		80:	// ABORTING
			// code that is executed only in the first cycle of this state
				IF xStateChange = TRUE THEN
					xStateChange := FALSE;
					iResponse := eResponseReadMalfunctionList.aborting;
					xBusy := FALSE;
					xDone := FALSE;
					xError := FALSE;
					xAborted := TRUE;
				END_IF
			//-----------------------------------------------------------------------------------------------------------
			
			// code that is repeated every cycle in this state
				IF iCurrentValveMode = 63 THEN
					iCommandNumber := 5;	// exit transfer mode
				ELSIF iCurrentValveMode <> 61 AND iCurrentValveMode <> 63 THEN
					iCommandNumber := 6;	// stop running motion apps
				ELSE
					iCommandNumber := 0; 
				END_IF
			//-----------------------------------------------------------------------------------------------------------
			
			// Transition
				IF xAbort = FALSE AND xExecute = FALSE AND iCurrentValveMode = 61 THEN
					xStateChange := TRUE;
					iState := 100;
				END_IF
			//-----------------------------------------------------------------------------------------------------------

		100:	// RESETTING FUNCTION BLOCK AND VALVE
			// code that is executed only in the first cycle of this state
				IF xStateChange = TRUE THEN
					xStateChange := FALSE;
					iResponse := eResponseReadMalfunctionList.resetting;
					xDone := FALSE;
					xError := FALSE;
					xBusy := FALSE;
					xAborted := FALSE;
					xFirstTransfer := FALSE;
				END_IF
			//-----------------------------------------------------------------------------------------------------------
			
			// code that is repeated every cycle in this state	
				IF iCurrentValveMode = 63 THEN
					iCommandNumber := 5;	// exit transfer mode
				ELSIF iCurrentValveMode <> 61 AND iCurrentValveMode <> 63 THEN
					iCommandNumber := 6;	// stop running motion apps
				END_IF
				
				FOR iCountMFLreset := 1 TO 40 BY 1 DO
					astMalfunctionlist[iCountMFLreset].usiMalfunctionCode := 0;
					astMalfunctionlist[iCountMFLreset].usiMalfunctionSubcode := 0;
					astMalfunctionlist[iCountMFLreset].usiMalfunctionClassification := 0;
				END_FOR
				
				iNumberOfMalfunctions := 0;
				iCountMFLreset := 0;
				iCountMFLdownload := 1;
				
			//-----------------------------------------------------------------------------------------------------------
			
			// Transition
				IF iCurrentValveMode = 61 THEN
					iCommandNumber := 6; // Last command to send before the FB is in IDLE
					xStateChange := TRUE;
					iState := 10;
				END_IF
			//-----------------------------------------------------------------------------------------------------------

		(*		
		00:	// ___STATE-TEMPLATE____
			// code that is executed only in the first cycle of this state
				IF xStateChange = TRUE THEN
					xStateChange := FALSE;
					eResponse := eTransferResponse.;
					xDone := ___;
					xError := ___;
					xBusy := ___;
					xAborted := ___;
				END_IF
			//-----------------------------------------------------------------------------------------------------------
			
			// code that is repeated every cycle in this state	
			//-----------------------------------------------------------------------------------------------------------
			
			// Transition
				IF ___ THEN
					xStateChange := TRUE;
					iState := 100;
				END_IF
			//-----------------------------------------------------------------------------------------------------------
			
		*)
		
	END_CASE
//-----------------------------------------------------------------------------------------------------------

// command section
	CASE iCommandNumber OF
		0:	// IDLE
		
		5:	// EXIT TRANSFER MODE
			fbwritevaluetoword(iValue:=63, iStartBit:=0, iEndBit:=5, wDataWord:=awBusDataToVTEM[0], xError=> );							// Valve Mode = 63
			fbwritevaluetoword(iValue:=0, iStartBit:=6, iEndBit:=7, wDataWord:=awBusDataToVTEM[0], xError=> );							// 0 (unused)
			fbwritevaluetoword(iValue:=0, iStartBit:=8, iEndBit:=12, wDataWord:=awBusDataToVTEM[0], xError=> );							// Channel = 0 (ignored)
			fbwritevaluetoword(iValue:=3, iStartBit:=13, iEndBit:=15, wDataWord:=awBusDataToVTEM[0], xError=> );						// Transfer Control = Exit transfer mode (3)
			fbwritevaluetoword(iValue:=0, iStartBit:=0, iEndBit:=7, wDataWord:=awBusDataToVTEM[1], xError=> );							// Addressed Target = 0 (ignored)
			fbwritevaluetoword(iValue:=0, iStartBit:=8, iEndBit:=15, wDataWord:=awBusDataToVTEM[1], xError=> );							// Index = 0 (ignored)
			fbwritevaluetoword(iValue:=0, iStartBit:=0, iEndBit:=15, wDataWord:=awBusDataToVTEM[2], xError=> );							// Value = 0 (ignored)
			
		6:	// stop running motion apps
			fbwritevaluetoword(iValue:=61, iStartBit:=0, iEndBit:=5, wDataWord:=awBusDataToVTEM[0], xError=> );							// Valve Mode = 61 (stop)
			fbwritevaluetoword(iValue:=0, iStartBit:=6, iEndBit:=7, wDataWord:=awBusDataToVTEM[0], xError=> );							// App Control = 0 (unused)
			fbwritevaluetoword(iValue:=0, iStartBit:=8, iEndBit:=15, wDataWord:=awBusDataToVTEM[0], xError=> );							// App Option = 0 (unused)
			fbwritevaluetoword(iValue:=0, iStartBit:=0, iEndBit:=15, wDataWord:=awBusDataToVTEM[1], xError=> );							// Setpoint Value 1 = 0 (unused)
			fbwritevaluetoword(iValue:=0, iStartBit:=0, iEndBit:=15, wDataWord:=awBusDataToVTEM[2], xError=> );							// Setpoint Value 2 = 0 (unused)
		
		10:	// getting count of malfunction messages
			fbwritevaluetoword(iValue:=63, iStartBit:=0, iEndBit:=5, wDataWord:=awBusDataToVTEM[0], xError=> );							// Valve Mode = 63 (transfer mode)
			fbwritevaluetoword(iValue:=31, iStartBit:=8, iEndBit:=12, wDataWord:=awBusDataToVTEM[0], xError=> );						// Channel = 31 (malfunctions)
			fbwritevaluetoword(iValue:=2, iStartBit:=13, iEndBit:=15, wDataWord:=awBusDataToVTEM[0], xError=> );						// Transfer Control = 2 (Upload)
			fbwritevaluetoword(iValue:=usiChooseOtherValve, iStartBit:=0, iEndBit:=7, wDataWord:=awBusDataToVTEM[1], xError=> );		// Addressed Target = usiChooseOtherValve
			fbwritevaluetoword(iValue:=255, iStartBit:=8, iEndBit:=15, wDataWord:=awBusDataToVTEM[1], xError=> );						// Index = 255 (Number of malfunction messages)
			fbwritevaluetoword(iValue:=0, iStartBit:=0, iEndBit:=15, wDataWord:=awBusDataToVTEM[2], xError=> );							// Value = 0 (Upload)
		
		40:	// reading malfunction list
			fbwritevaluetoword(iValue:=63, iStartBit:=0, iEndBit:=5, wDataWord:=awBusDataToVTEM[0], xError=> );							// Valve Mode = 63 (transfer mode)
			fbwritevaluetoword(iValue:=31, iStartBit:=8, iEndBit:=12, wDataWord:=awBusDataToVTEM[0], xError=> );						// Channel = 31 (malfunctions)
			fbwritevaluetoword(iValue:=2, iStartBit:=13, iEndBit:=15, wDataWord:=awBusDataToVTEM[0], xError=> );						// Transfer Control = 2 (Upload)
			fbwritevaluetoword(iValue:=usiChooseOtherValve, iStartBit:=0, iEndBit:=7, wDataWord:=awBusDataToVTEM[1], xError=> );		// Addressed Target = usiChooseOtherValve
			fbwritevaluetoword(iValue:=iCountMFLdownload, iStartBit:=8, iEndBit:=15, wDataWord:=awBusDataToVTEM[1], xError=> );			// Index = iCounterMFLdownload (Number of malfunction messages)
			fbwritevaluetoword(iValue:=0, iStartBit:=0, iEndBit:=15, wDataWord:=awBusDataToVTEM[2], xError=> );							// Value = 0 (Upload)

	END_CASE	
//-----------------------------------------------------------------------------------------------------------

END_FUNCTION_BLOCK

// Transfermode/specific_MA_config/FB_Write_config_MA_10
// This function block can be used to download the configuration of Motion App 10 ("Flow control").
// The specific parameters of this Motion App are the inputs of this FB and can be defined by the user. 
// The function block uses the transfer mode to write this configuration to the Motion Terminal
// and indicates the state of the download process.

FUNCTION_BLOCK FB_Write_config_MA_10
VAR_INPUT
	awBusDataFromVTEM 				: ARRAY [0..2] OF WORD;		(* 6 bytes of process data received from the Motion Terminal *)
END_VAR
	
VAR_IN_OUT
	awBusDataToVTEM 				: ARRAY [0..2] OF WORD; 	(* 6 bytes of process data sent to the Motion Terminal *)
END_VAR

VAR_INPUT
	xExecute 						: BOOL; 					(* has to be set to TRUE for a download and to FALSE to reset the function block after a download *)

	iParameterSet					: INT := 1; 				(* the parameter set to be written to, 1 by default *)
	
	// system parameters
		iOperatingMedium			: eMA10OperatingMedium := 1;// Type and condition of the operating medium (values see eMA10OperatingMedium)
		iInPortFlowRate2_optional	: INT;						// Sensor port for flow rate at (2) (required for closed-loop controlled operating mode, value is number of the slot (beginning from 0 and including valve slots) * 10 + number of the port 
		iInPortFlowRate4_optional	: INT;						// Sensor port for flow rate at (4) (required for closed-loop controlled operating mode, value is number of the slot (beginning from 0 and including valve slots) * 10 + number of the port
		iInPortRetracted_optional	: INT;						// Sensor port for detection of end position at pressurisation of outlet port 2 (retracted), value is number of the slot (beginning from 0 and including valve slots) * 10 + number of the port
		iInPortAdvanced_optional	: INT;						// Sensor port for detection of end position at pressurisation of outlet port 4 (advanced), value is number of the slot (beginning from 0 and including valve slots) * 10 + number of the port

	// application parameters
		iCharacteristicAt2			: INT;						// Control characteristic, outlet port (2) (0 = "fast" (short tubes), 1 = medium (medium length tubes), 2 = "universal" (esp. long tubes), 3 = defined by tuning parameters (only if closed-loop control is activated for outlet port (2)))
		iCharacteristicAt4			: INT;						// Control characteristic, outlet port (4) (0 = "fast" (short tubes), 1 = medium (medium length tubes), 2 = "universal" (esp. long tubes), 3 = defined by tuning parameters (only if closed-loop control is activated for outlet port (4)))
		xClosedLoopControl2			: BOOL := FALSE;			// TRUE acivates closed-loop control for outlet port (2), FALSE ist open-loop controlled operation
		xClosedLoopControl4			: BOOL := FALSE;			// TRUE acivates closed-loop control for outlet port (4), FALSE ist open-loop controlled operation
		
	// tuning parameters
		iOptProportionalGainFor2	: INT;						// Optional tuning parameter for the customized proportional element of the PID modulator at outlet port (2) [1 digit = 0.01 g/s/bar]
		iOptIntegralGainFor2		: INT;						// Optional tuning parameter for the customized integral element of the PID modulator at outlet port (2) [1 digit = 0.01 g/s²/bar]
		iOptRedFeedforwContrRate2	: INT;						// Optional tuning parameter for reduction of feedforward control rate of 100% for outlet port (2) [1 digit = 1%]
		iOptBoostSetpointReach2		: INT;						// Optional tuning parameter for boost to reach the setpoint value for outlet port (2) earlier, but with higher overshoot [1 digit = 1%] 
		iOptOffsetTargFRLimitInfo2	: INT;						// Optional tuning parameter for offset on the threshold value of 95% of the possible relative flow at outlet port (2) for feedback in app state, bit 5 [1 digit = 1%]
		iOptOffsetMinConsSetp2		: INT;						// Optional tuning parameter for offset to the threshold value of 25 l/min, below which a target flow rate for outlet port (2) is not considered [1 digit = 1 l/min]

		iOptProportionalGainFor4	: INT;						// Optional tuning parameter for the customized proportional element of the PID modulator at outlet port (4) [1 digit = 0.01 g/s/bar]
		iOptIntegralGainFor4		: INT;						// Optional tuning parameter for the customized integral element of the PID modulator at outlet port (4) [1 digit = 0.01 g/s²/bar]
		iOptRedFeedforwContrRate4	: INT;						// Optional tuning parameter for reduction of feedforward control rate of 100% for outlet port (4) [1 digit = 1%]
		iOptBoostSetpointReach4		: INT;						// Optional tuning parameter for boost to reach the setpoint value for outlet port (4) earlier, but with higher overshoot [1 digit = 1%] 
		iOptOffsetTargFRLimitInfo4	: INT;						// Optional tuning parameter for offset on the threshold value of 95% of the possible relative flow at outlet port (4) for feedback in app state, bit 5 [1 digit = 1%]
		iOptOffsetMinConsSetp4		: INT;						// Optional tuning parameter for offset to the threshold value of 25 l/min, below which a target flow rate for outlet port (4) is not considered [1 digit = 1 l/min]
END_VAR

VAR_OUTPUT                  		
	iResponse 						: eTransferResponse; 		(* returns the status of the execution of the download process *)
	sCurrentValue 					: STRING; 					(* indicates which value of the array is currently treated (necessary to evaluate in case of error messages) *)
	xDownloadDone 					: BOOL; 					(* indicates whether the download was successful *)
	xDownloadError 					: BOOL := FALSE; 			(* indicates whether an error occurred during the transfer *)
END_VAR

VAR
	aTransferPackages				: ARRAY [0..100] OF stTransferPackage;
	fbdownloadMultipleParameters 	: FB_Download_Multiple_Parameters;
	iCurrentValue					: INT;
	fbWriteValueToWord 				: FB_Write_Value_To_Word;
	iOperatingMode					: INT;						// Container for the information of the variables xClosedLoopControl2 and xClosedLoopControl4
	wOperatingMode					: WORD;						// word container for the operating mode
END_VAR

(*****************************************************************************************************

Festo SE & Co. KG, Esslingen
Copyright (c) 2020. All rights reserved.

Product:            Motion Terminal VTEM
Description:        Function Block to download the parameters for Motion App 10 to the Motion Terminal

Object version:     1.00
Last change:        2021-02
======================================================================================================
                                       H I S T O R Y
======================================================================================================
Version:            1.00
Date:               2021-02
Change/Activity:    - created (#3805775)
Release:            3.5.7.236 (CODESYS 3.5.7.2, Lib version 3.6)
Author:             JEBU
======================================================================================================

*****************************************************************************************************)

// combine xClosedLoopControl2 and xClosedLoopControl4 into iOperatingMode (Bit 0 = (4), Bit 1 = (2))
	wOperatingMode.0 := xClosedLoopControl4;
	wOperatingMode.1 := xClosedLoopControl2; 
	iOperatingMode := WORD_TO_INT(wOperatingMode);

// write the Motion App specific parameters into the struct
	//iOperatingMedium
		aTransferPackages[0].iChannel := iParameterSet;
		aTransferPackages[0].iAddressedTarget := 10;
		aTransferPackages[0].iIndex := 42;
		aTransferPackages[0].iTransferValue := iOperatingMedium;
	
	//iInPortFlowRate2_optional
		aTransferPackages[1].iChannel := iParameterSet;
		aTransferPackages[1].iAddressedTarget := 10;
		aTransferPackages[1].iIndex := 81;
		aTransferPackages[1].iTransferValue := iInPortFlowRate2_optional;

	//iInPortFlowRate4_optional
		aTransferPackages[2].iChannel := iParameterSet;
		aTransferPackages[2].iAddressedTarget := 10;
		aTransferPackages[2].iIndex := 82;
		aTransferPackages[2].iTransferValue := iInPortFlowRate4_optional;
	
	//iInPortRetracted_optional
		aTransferPackages[3].iChannel := iParameterSet;
		aTransferPackages[3].iAddressedTarget := 10;
		aTransferPackages[3].iIndex := 70;
		aTransferPackages[3].iTransferValue := iInPortRetracted_optional;
	
	//iInPortAdvanced_optional
		aTransferPackages[4].iChannel := iParameterSet;
		aTransferPackages[4].iAddressedTarget := 10;
		aTransferPackages[4].iIndex := 71;
		aTransferPackages[4].iTransferValue := iInPortAdvanced_optional;
	
	//iCharacteristicAt2
		aTransferPackages[5].iChannel := iParameterSet;
		aTransferPackages[5].iAddressedTarget := 10;
		aTransferPackages[5].iIndex := 220;
		aTransferPackages[5].iTransferValue := iCharacteristicAt2;
	
	//iCharacteristicAt4
		aTransferPackages[6].iChannel := iParameterSet;
		aTransferPackages[6].iAddressedTarget := 10;
		aTransferPackages[6].iIndex := 221;
		aTransferPackages[6].iTransferValue := iCharacteristicAt4;
	
	//iOperatingMode
		aTransferPackages[7].iChannel := iParameterSet;
		aTransferPackages[7].iAddressedTarget := 10;
		aTransferPackages[7].iIndex := 223;
		aTransferPackages[7].iTransferValue := iOperatingMode;
	
	//iOptProportionalGainFor2
		aTransferPackages[8].iChannel := iParameterSet;
		aTransferPackages[8].iAddressedTarget := 10;
		aTransferPackages[8].iIndex := 230;
		aTransferPackages[8].iTransferValue := iOptProportionalGainFor2;
	
	//iOptIntegralGainFor2
		aTransferPackages[9].iChannel := iParameterSet;
		aTransferPackages[9].iAddressedTarget := 10;
		aTransferPackages[9].iIndex := 231;
		aTransferPackages[9].iTransferValue := iOptIntegralGainFor2;
	
	//iOptRedFeedforwContrRate2
		aTransferPackages[10].iChannel := iParameterSet;
		aTransferPackages[10].iAddressedTarget := 10;
		aTransferPackages[10].iIndex := 232;
		aTransferPackages[10].iTransferValue := iOptRedFeedforwContrRate2;
	
	//iOptBoostSetpointReach2
		aTransferPackages[11].iChannel := iParameterSet;
		aTransferPackages[11].iAddressedTarget := 10;
		aTransferPackages[11].iIndex := 233;
		aTransferPackages[11].iTransferValue := iOptBoostSetpointReach2;
	
	//iOptOffsetTargFRLimitInfo2
		aTransferPackages[12].iChannel := iParameterSet;
		aTransferPackages[12].iAddressedTarget := 10;
		aTransferPackages[12].iIndex := 234;
		aTransferPackages[12].iTransferValue := iOptOffsetTargFRLimitInfo2;
	
	//iOptOffsetMinConsSetp2
		aTransferPackages[13].iChannel := iParameterSet;
		aTransferPackages[13].iAddressedTarget := 10;
		aTransferPackages[13].iIndex := 235;
		aTransferPackages[13].iTransferValue := iOptOffsetMinConsSetp2;
	
	//iOptProportionalGainFor4
		aTransferPackages[14].iChannel := iParameterSet;
		aTransferPackages[14].iAddressedTarget := 10;
		aTransferPackages[14].iIndex := 240;
		aTransferPackages[14].iTransferValue := iOptProportionalGainFor4;
	
	//iOptIntegralGainFor4
		aTransferPackages[15].iChannel := iParameterSet;
		aTransferPackages[15].iAddressedTarget := 10;
		aTransferPackages[15].iIndex := 241;
		aTransferPackages[15].iTransferValue := iOptIntegralGainFor4;
	
	//iOptRedFeedforwContrRate4
		aTransferPackages[16].iChannel := iParameterSet;
		aTransferPackages[16].iAddressedTarget := 10;
		aTransferPackages[16].iIndex := 242;
		aTransferPackages[16].iTransferValue := iOptRedFeedforwContrRate4;
	
	//iOptBoostSetpointReach4
		aTransferPackages[17].iChannel := iParameterSet;
		aTransferPackages[17].iAddressedTarget := 10;
		aTransferPackages[17].iIndex := 243;
		aTransferPackages[17].iTransferValue := iOptBoostSetpointReach4;
	
	//iOptOffsetTargFRLimitInfo4
		aTransferPackages[18].iChannel := iParameterSet;
		aTransferPackages[18].iAddressedTarget := 10;
		aTransferPackages[18].iIndex := 244;
		aTransferPackages[18].iTransferValue := iOptOffsetTargFRLimitInfo4;
	
	//iOptOffsetMinConsSetp4
		aTransferPackages[19].iChannel := iParameterSet;
		aTransferPackages[19].iAddressedTarget := 10;
		aTransferPackages[19].iIndex := 245;
		aTransferPackages[19].iTransferValue := iOptOffsetMinConsSetp4;
	
	// define end of parameter list to be downloaded by setting all variables to 0 (end criterion for FB_Download_Multiple_Parameters)
		aTransferPackages[20].iChannel := 0;
		aTransferPackages[20].iAddressedTarget := 0;
		aTransferPackages[20].iIndex := 0;
		aTransferPackages[20].iTransferValue := 0;


// pre-check of the value for the parameter set
	IF xExecute = TRUE AND (iParameterSet < 1 OR iParameterSet > 5) THEN		// invalid input for the parameter set
		xDownloadDone := FALSE; 
		xDownloadError := TRUE; 
		iResponse := eTransferResponse.invalid_ParameterSet; 
		iCurrentValue := 0; 
		// send command 'stop'
		fbWriteValueToWord(iValue := 61, iStartBit := 0, iEndBit := 5, wDataWord := awBusDataToVTEM[0]); 			// ValveMode = 61
		fbWriteValueToWord(iValue := 0, iStartBit := 6, iEndBit := 15, wDataWord := awBusDataToVTEM[0]); 			// (empty)
		awBusDataToVTEM[1] := 0; 
		awBusDataToVTEM[2] := 0; 
		
	ELSE	
		// call the function block for multiple parameter download
			fbdownloadMultipleParameters(	xExecute := xExecute,
											awBusDataFromVTEM := awBusDataFromVTEM,
											aTransferPackages := aTransferPackages, 
											awBusDataToVTEM := awBusDataToVTEM,
											xDownloadDone => xDownloadDone,
											xDownloadError => xDownloadError,
											iResponse => iResponse,
											iCurrentValue => iCurrentValue);
	END_IF
	
	
// The current value output is needed if there is any invalid value in order to address it correctly.
// As the user doesn't work with indices in this function block, the current value is transformed to a string holding the name of the parameter.
	CASE iCurrentValue OF
		0: sCurrentValue := 'iOperatingMedium';
		1: sCurrentValue := 'iInPortFlowRate2_optional';
		2: sCurrentValue := 'iInPortFlowRate4_optional';
		3: sCurrentValue := 'iInPortRetracted_optional';
		4: sCurrentValue := 'iInPortAdvanced_optional';
		5: sCurrentValue := 'iCharacteristicAt2';
		6: sCurrentValue := 'iCharacteristicAt4';
		7: sCurrentValue := 'iOperatingMode';
		8: sCurrentValue := 'iOptProportionalGainFor2';
		9: sCurrentValue := 'iOptIntegralGainFor2';
		10: sCurrentValue := 'iOptRedFeedforwContrRate2';
		11: sCurrentValue := 'iOptBoostSetpointReach2';
		12: sCurrentValue := 'iOptOffsetTargFRLimitInfo2';
		13: sCurrentValue := 'iOptOffsetMinConsSetp2';
		14: sCurrentValue := 'iOptProportionalGainFor4';
		15: sCurrentValue := 'iOptIntegralGainFor4';
		16: sCurrentValue := 'iOptRedFeedforwContrRate4';
		17: sCurrentValue := 'iOptBoostSetpointReach4';
		18: sCurrentValue := 'iOptOffsetTargFRLimitInfo4';
		19: sCurrentValue := 'iOptOffsetMinConsSetp4';
		20: sCurrentValue := 'AllParametersWritten';
	END_CASE

END_FUNCTION_BLOCK

// StateInterpreter/FB_StateInterpreter_MA_10
/// The variable "byActualAppState" is an output of the FB_ValveControl that is used differently in each Motion App.
/// This function block interprets the "AppState" output of the FB_ValveControl if Motion App 10 ("Flow control") is running.
/// The Motion App specific values are derived from the "byActualAppState".

FUNCTION_BLOCK FB_StateInterpreter_MA_10
VAR_INPUT
	byActualAppState 			: BYTE; 	(* output of the FB_ValveControl *)
END_VAR
VAR_OUTPUT
	x2or4outOfSpec				: BOOL;		// indicates that port (2) and/or (4) is operated outside the specification
	xFlow2FromMeasurement		: BOOL;		// indicates that actual value for flow on (2) comes from measurement (higher accuracy)
	xFlow4FromMeasurement		: BOOL;		// indicates that actual value for flow on (4) comes from measurement (higher accuracy)
	xRatioSetToMaxOverLimit2	: BOOL;		// Indicates that the ratio of the set flow to the maximum adjustable flow at port (2) is greater than the specified limit (95% of the maximum adjustable flow + value of parameter "iOptOffsetTargFRLimitInfo2")
	xRatioSetToMaxOverLimit4	: BOOL;		// Indicates that the ratio of the set flow to the maximum adjustable flow at port (4) is greater than the specified limit (95% of the maximum adjustable flow + value of parameter "iOptOffsetTargFRLimitInfo4")
	xRetractedEndPos_optional	: BOOL;  	(* only if digital sensors are installed (optional): indicates whether the retracted end position was reached (after outlet port 2 is pressurised) *)
	xAdvancedEndPos_optional	: BOOL;  	(* only if digital sensors are installed (optional): indicates whether the advanced end position was reached (after outlet port 4 is pressurised) *)
	xWarning					: BOOL; 	(* indicates whether there is a warning returned by the Motion App *)
END_VAR
VAR
	fbReadBitsFromByte			: FB_Read_Bits_From_Byte;
	by2or4outOfSpec				: BYTE;
	byFlow2FromMeasurement		: BYTE;	
	byFlow4FromMeasurement		: BYTE;	
	byRatioSetToMaxOverLimit2	: BYTE;	
	byRatioSetToMaxOverLimit4	: BYTE;
	byRetractedEndPos			: BYTE;
	byAdvancedEndPos			: BYTE;
	byWarning					: BYTE;
END_VAR

(*****************************************************************************************************

Festo SE & Co. KG, Esslingen
Copyright (c) 2020. All rights reserved.

Product:            Motion Terminal VTEM
Description:        Function block for interpreting the app state of Motion App 10 

Object version:     1.00
Last change:        2020-11
======================================================================================================
                                       H I S T O R Y
======================================================================================================
Version:            1.00
Date:               2020-11
Change/Activity:    - created (#3805730)
Release:            3.5.7.236
Author:             JEBU
======================================================================================================

*****************************************************************************************************)

// read the Motion App specific values from the ActualAppState byte
fbReadBitsFromByte(byData := byActualAppState, iStartBit := 1, iEndBit := 1, byValue => by2or4outOfSpec);
x2or4outOfSpec :=  BYTE_TO_BIT(by2or4outOfSpec);

fbReadBitsFromByte(byData := byActualAppState, iStartBit := 3, iEndBit := 3, byValue => byFlow2FromMeasurement);
xFlow2FromMeasurement :=  BYTE_TO_BIT(byFlow2FromMeasurement);

fbReadBitsFromByte(byData := byActualAppState, iStartBit := 4, iEndBit := 4, byValue => byFlow4FromMeasurement);
xFlow4FromMeasurement :=  BYTE_TO_BIT(byFlow4FromMeasurement);

fbReadBitsFromByte(byData := byActualAppState, iStartBit := 5, iEndBit := 5, byValue => byRatioSetToMaxOverLimit2);
xRatioSetToMaxOverLimit2 :=  BYTE_TO_BIT(byRatioSetToMaxOverLimit2);

fbReadBitsFromByte(byData := byActualAppState, iStartBit := 6, iEndBit := 6, byValue => byRatioSetToMaxOverLimit4);
xRatioSetToMaxOverLimit4 :=  BYTE_TO_BIT(byRatioSetToMaxOverLimit4);

fbReadBitsFromByte(byData := byActualAppState, iStartBit := 0, iEndBit := 0, byValue => byRetractedEndPos);
xRetractedEndPos_optional :=  BYTE_TO_BIT(byRetractedEndPos);

fbReadBitsFromByte(byData := byActualAppState, iStartBit := 2, iEndBit := 2, byValue => byAdvancedEndPos); 
xAdvancedEndPos_optional :=  BYTE_TO_BIT(byAdvancedEndPos);

fbReadBitsFromByte(byData := byActualAppState, iStartBit := 7, iEndBit := 7, byValue => byWarning);
xWarning := BYTE_TO_BIT(byWarning);

END_FUNCTION_BLOCK

// Operation/FB_AppOptionGenerator_MA_02
/// The App Option byte of Motion App 02 ("Proportional directional control valve") contains several pieces of information.
/// The individual pieces of information can be passed to this function block and it generates the corresponding value for the App Option byte from this.
/// The generated App Option byte can be passed to the FB_ValveControl block.

FUNCTION_BLOCK FB_AppOptionGenerator_MA_02
VAR_INPUT
	usiValveType			: USINT;		// Defines used valve type (14 = 4/3 G (normally closed), 15 = 2 × 3/3nG (normally closed))
	xSetMeaningOfActVal1	: BOOL;			// Setting the meaning of actual value 1 (0 = valve position, 1 = relative pressure)
	xSetMeaningOfActVal2	: BOOL;			// Setting the meaning of actual value 2 (0 = valve position, 1 = relative pressure)
END_VAR
VAR_OUTPUT
	byAppOption				: BYTE;			// AppOption byte to connect with the byAppOption input of FB_ValveControl
END_VAR
VAR
END_VAR

(*****************************************************************************************************

Festo SE & Co. KG, Esslingen
Copyright (c) 2021. All rights reserved.

Product:            Motion Terminal VTEM
Description:        Function block for generating the app option byte for Motion App 2

Object version:     1.00
Last change:        2021-01
======================================================================================================
                                       H I S T O R Y
======================================================================================================
Version:            1.00
Date:               2021-01
Change/Activity:    - created (#3919898)
Release:            3.5.7.236
Author:             JEBU
======================================================================================================

*****************************************************************************************************)
IF usiValveType >= 14 AND usiValveType <= 15 THEN
	byAppOption := USINT_TO_BYTE(usiValveType);
	byAppOption.5 := xSetMeaningOfActVal1;
	byAppOption.6 := xSetMeaningOfActVal2;	
ELSE
	byAppOption := 0;
END_IF

END_FUNCTION_BLOCK
